TEXTLIST TextList_FootPedalerroid
  0 = 'no_error'
  1 = 'not_connected'
  2 = 'invalid_state'
  3 = 'io_error'
  4 = 'unknown_error'
  666 = 'emergency_error'
   = ''
END_TEXTLIST

(* stored: Version 1.1.0.1, ProductVersion 3.1.4024.11
   TextList TextList_FootPedalerroid: Id {196e29f5-29d0-4e68-a78f-2e20dec27182} *)
